{attribute 'linkalways'} 
{attribute 'no_explicit_call' := 'This FB is a CLASS and must be accessed using methods or properties'}
{attribute 'enable_dynamic_creation'}
FUNCTION_BLOCK _INT EXTENDS DatatypeBase
VAR
	localData : INT;
	activeData : REFERENCE TO INT REF= localData;
END_VAR

PROPERTY PUBLIC Address : PVOID
GET
Address := ADR(activeData);
END_GET
END_PROPERTY

METHOD PUBLIC ClearReference
VAR_INPUT
END_VAR
activeData REF= localData;
END_METHOD

METHOD PUBLIC Clone : I_Datatype
VAR
    pClone : POINTER TO _INT;
END_VAR
pClone := __NEW(_INT(InitialValue := Value));
Clone := pClone^;
END_METHOD

METHOD FB_init : BOOL
VAR_INPUT
	bInitRetains : BOOL; // if TRUE, the retain variables are initialized (warm start / cold start)
	bInCopyCode : BOOL;  // if TRUE, the instance afterwards gets moved into the copy code (online change)
	InitialValue : INT;
END_VAR
localData := InitialValue;
END_METHOD

PROPERTY PUBLIC Identifier : T_MAXSTRING
GET
Identifier := 'INT';
END_GET
END_PROPERTY

PROPERTY PUBLIC IecType : T_MAXSTRING
GET
IecType := 'INT';
END_GET
END_PROPERTY

METHOD PUBLIC ReferenceOf
VAR_INPUT
	ReferenceTarget : INT;
END_VAR
activeData REF= ReferenceTarget;
END_METHOD

METHOD PUBLIC SerializeWith
VAR_INPUT
	Serializer : I_Serializer;
END_VAR
Serializer.AddInt(activeData);
END_METHOD

PROPERTY PUBLIC Size : UDINT
GET
Size := SIZEOF(activeData);
END_GET
END_PROPERTY

METHOD TryDeserializeFrom : BOOL
VAR_INPUT
	Deserializer : I_Deserializer;
END_VAR
TryDeserializeFrom := Deserializer.TryGetInt(activeData);
END_METHOD

METHOD TryMakeReferenceOf : BOOL
VAR_INPUT
	Target : I_Datatype;
END_VAR
VAR
	pTargetData : POINTER TO INT;
END_VAR
IF NOT (Target.Identifier = Identifier) THEN
	RETURN;
END_IF

pTargetData := Target.Address;
activeData REF= pTargetData^;
TryMakeReferenceOf := TRUE;
END_METHOD

PROPERTY PUBLIC Value : INT
GET
Value := activeData;
END_GET
SET
activeData := Value;
END_SET
END_PROPERTY

END_FUNCTION_BLOCK

(* stored: Version 1.1.0.1, ProductVersion 3.1.4024.12
   POU _INT: Id {e1db94ec-2dc4-44cc-ade8-bd509d56f134}, SpecialFunc None
   Folder Constructor: Id {e6663295-a004-4cd8-9b8e-ba3c80dc3fca}
   Property Address: Id {d9f4f2d6-a451-4f3d-b399-675ccf7ce1e9}
   Get Get: Id {5087d04c-b7e8-4d27-83ce-93f6edba9c30}
   Method ClearReference: Id {a9971519-22ed-418b-b2f3-223dbf639d4f}
   Method Clone: Id {37c85a4c-3715-45a4-affe-5676fdc946c4}
   Method FB_init: Id {9f83609a-a42c-45f4-a3c3-c95a48d82e7e}
   Property Identifier: Id {803cba95-d958-4e03-a926-d5adf0c86fe5}
   Get Get: Id {f20cfaef-4a0f-4a36-8dbe-c8bccec1599f}
   Property IecType: Id {93df8d16-361c-0589-1f02-56441476a1c3}
   Get Get: Id {e4478699-f245-0f2c-0325-791fec8c3d09}
   Method ReferenceOf: Id {10808909-7a1b-0eae-399d-be00cd1ce852}
   Method SerializeWith: Id {78bbb435-9f2e-431a-8b4c-405d57f91cbd}
   Property Size: Id {31acef3f-a1c0-4d9a-bcfb-ca14a4a2b491}
   Get Get: Id {23c38faf-f22a-43f5-a149-f7f4a03bec90}
   Method TryDeserializeFrom: Id {69d264a8-dbe3-48fa-a85c-7902fb2ef2a8}
   Method TryMakeReferenceOf: Id {9c0d1585-3764-49dd-8abd-c30f2cd927f2}
   Property Value: Id {a7292d94-0f0c-4318-b80c-30f7fa487b67}
   Get Get: Id {273173e7-de92-441f-b4c2-5d1ca742f0a3}
   Set Set: Id {d0072a17-05b1-4caf-bb6f-903572100699} *)
